DATA_BLOCK "DB_PlcDiagnosticsModel"
{ S7_Optimized_Access := 'TRUE' }
VERSION : 0.1
NON_RETAIN
   VAR
      Data : "UDT_PlcDiagnosticsModel";
   END_VAR

BEGIN
END_DATA_BLOCK
